{attribute 'qualified_only'}
VAR_GLOBAL
	iVar AT%M*    : INT;
	bVar AT%M*	  : BOOL;
END_VAR

(* stored: Version 1.1.0.1, ProductVersion 3.1.4024.12
   GVL GVL_ADS: Id {6fece0e0-2ae2-48a3-ae3a-e51fc2c8d25f} *)
